FUNCTION_BLOCK TUnsupportedEventHandler IMPLEMENTS IUnsupportedEventHandler
VAR_INPUT
END_VAR
VAR_OUTPUT
END_VAR
VAR
END_VAR

END_FUNCTION_BLOCK

(* stored: Version 1.1.0.1, ProductVersion 3.1.4024.3
   POU TUnsupportedEventHandler: Id {9c2e5d32-b5a9-43b0-b18a-e8571f4432bb}, SpecialFunc None *)
